// TIA Portal V17 program export: 1 tag tables, 0 data types, 2 data blocks, 2 code blocks (in call order from the OBs), 3 instance data blocks

VAR_GLOBAL   // PLC tag table "Default tag table"
   clockInput AT %I0.0 : Bool;   // Clock generator input
   Tag_1 AT %ID1000 : DWord;
   Axe_1_Signal_A AT %Q0.2 : Bool;
   Axe_1_Signal_B AT %Q0.3 : Bool;
END_VAR

DATA_BLOCK "DataExample1"   // DB1
{ S7_Optimized_Access := 'TRUE' }
VERSION : 0.1
// stored: AutoNumber true, DBAccessibleFromOPCUA true, IsOnlyStoredInLoadMemory false, IsRetainMemResEnabled false, IsWriteProtectedInAS false, MemoryReserve 100
   VAR
      hscData { S7_SetPoint := 'True'} : HSC_Period;   // Instruction CTRL_HSC_EXT: CTRL
      hscDone : Bool;   // Instruction CTRL_HSC_EXT: Done
      hscBusy : Bool;   // Instruction CTRL_HSC_EXT: Busy
      hscError : Bool;   // Instruction CTRL_HSC_EXT: Error
      hscStatus : Word;   // Instruction CTRL_HSC_EXT: Status
      numPulsePerRot : Int := 1000;   // Number of pulses per rotation
      overflow : Bool;   // Elapsed time overflow
      speed : Real := 0.0;   // Calculated speed [rpm]
      vitesse : Real;
   END_VAR
BEGIN
   hscData.EnHSC := TRUE;
   hscData.NewPeriod := 10;
END_DATA_BLOCK

DATA_BLOCK "DataExample2"   // DB5
{ S7_Optimized_Access := 'TRUE' }
VERSION : 0.1
// stored: AutoNumber false, DBAccessibleFromOPCUA true, IsOnlyStoredInLoadMemory false, IsRetainMemResEnabled false, IsWriteProtectedInAS false, MemoryReserve 100
   VAR
      hscData { S7_SetPoint := 'True'} : HSC_Period;   // Instruction CTRL_HSC_EXT: CTRL
      hscDone : Bool;   // Instruction CTRL_HSC_EXT: Done
      hscBusy : Bool;   // Instruction CTRL_HSC_EXT: Busy
      hscError : Bool;   // Instruction CTRL_HSC_EXT: Error
      hscStatus : Word;   // Instruction CTRL_HSC_EXT: Status
      numPulsePerRot : Int := 1000;   // Number of pulses per rotation
      overflow : Bool;   // Elapsed time overflow
      speed : Real := 0.0;   // Calculated speed [rpm]
      vitesse : Real;
      hsc1 : HSC_Count;
   END_VAR
BEGIN
   hscData.EnHSC := TRUE;
   hscData.NewPeriod := 10;
END_DATA_BLOCK

ORGANIZATION_BLOCK "Main"   // OB1, FBD, ProgramCycle
TITLE = "Main Program Sweep (Cycle)"
{ S7_Optimized_Access := 'TRUE' }
VERSION : 0.1
// stored: AutoNumber true, IsIECCheckEnabled false, SetENOAutomatically false
   VAR_INPUT
      Initial_Call : Bool;   // Initial call of this OB
      Remanence : Bool;   // =True, if remanent data are available
   END_VAR
BEGIN

REGION Network 1: Call CTRL_HSC_EXT for HSC1
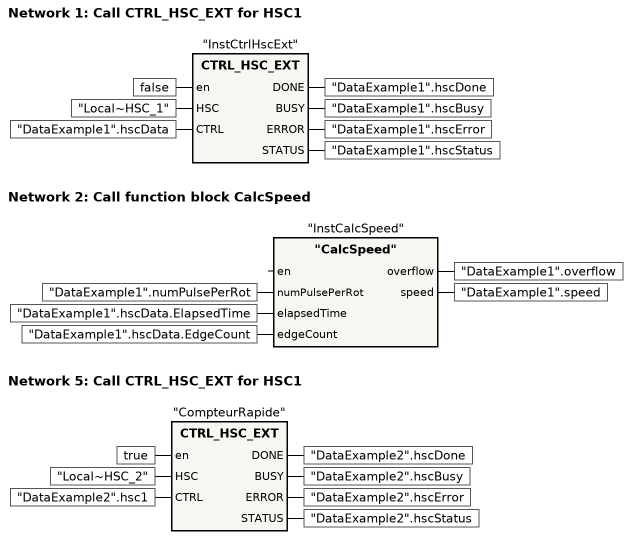
   IF false THEN
       "InstCtrlHscExt"(HSC := "Local~HSC_1",   // CTRL_HSC_EXT
                        CTRL := "DataExample1".hscData,
                        DONE => "DataExample1".hscDone,
                        BUSY => "DataExample1".hscBusy,
                        ERROR => "DataExample1".hscError,
                        STATUS => "DataExample1".hscStatus);
   END_IF;
END_REGION

REGION Network 2: Call function block CalcSpeed
   "InstCalcSpeed"(numPulsePerRot := "DataExample1".numPulsePerRot,   // "CalcSpeed"
                   elapsedTime := "DataExample1".hscData.ElapsedTime,
                   edgeCount := "DataExample1".hscData.EdgeCount,
                   overflow => "DataExample1".overflow,
                   speed => "DataExample1".speed);
END_REGION

REGION Network 3 (SCL)
   "DataExample1".vitesse := 0.2 * "DataExample1".speed;
END_REGION

REGION Network 5: Call CTRL_HSC_EXT for HSC1
   IF true THEN
       "CompteurRapide"(HSC := "Local~HSC_2",   // CTRL_HSC_EXT
                        CTRL := "DataExample2".hsc1,
                        DONE => "DataExample2".hscDone,
                        BUSY => "DataExample2".hscBusy,
                        ERROR => "DataExample2".hscError,
                        STATUS => "DataExample2".hscStatus);
   END_IF;
END_REGION
END_ORGANIZATION_BLOCK

FUNCTION_BLOCK "CalcSpeed"
{ S7_Optimized_Access := 'TRUE' }
VERSION : 0.1
   VAR_INPUT 
      numPulsePerRot : Int;
      elapsedTime { ExternalAccessible := 'False'; ExternalVisible := 'False'; ExternalWritable := 'False'} : UDInt;
      edgeCount { ExternalAccessible := 'False'; ExternalVisible := 'False'; ExternalWritable := 'False'} : UDInt;
   END_VAR

   VAR_OUTPUT 
      overflow { ExternalWritable := 'False'} : Bool;
      speed { ExternalWritable := 'False'} : Real;
   END_VAR

   VAR 
      statPeriod { ExternalAccessible := 'False'; ExternalVisible := 'False'; ExternalWritable := 'False'} : Real;
      statOverflow { ExternalAccessible := 'False'; ExternalVisible := 'False'; ExternalWritable := 'False'} : Bool;
   END_VAR

   VAR CONSTANT 
      BILLION : Real := 1.0E+09;
      OVERFLOW_VALUE : UDInt := 4294967295;
   END_VAR


BEGIN
	//=============================================================================
	//SIEMENS AG
	//(c)Copyright 2016 All Rights Reserved
	//-----------------------------------------------------------------------------
	//Library:       -
	//Tested with:   S7-1200 V4.2
	//Engineering:   TIA Portal V14
	//Restrictions:  -
	//Requirements:  S7-1200
	//Functionality: Basic axis functions, as power, reset, home and jog
	//-----------------------------------------------------------------------------
	//Change log table:
	//Version  Date       Expert in charge Changes applied
	//01.00.00 09.11.2016 Online Support   First released version
	//=============================================================================
	
	// #elapsedTime (range): 0 to 4.294.967.280
	// #elapsedTime (overflow): 4.294.967.295 (0xFFFF FFFF)
	
	// If EdgeCount and ElapsedTime is valid, calculate the period
	IF (#edgeCount > 0)
	  AND (#elapsedTime > 0)
	  AND (#elapsedTime <= 4294967280)
	THEN
	  // Calculate the period in nanoseconds 
	  #statPeriod := #elapsedTime / #edgeCount;
	  // Calculate the period in seconds 
	  #statPeriod := #numPulsePerRot * #statPeriod / #BILLION;
	END_IF;
	
	// Check overflow (the period between two pulse edges exceeds 4.295 seconds)
	IF (#elapsedTime = #OVERFLOW_VALUE)
	THEN
	  #statOverflow := TRUE;
	ELSE
	  #statOverflow := FALSE;
	END_IF;
	
	// Set period to zero, if overflow
	IF(#statOverflow = TRUE)
	THEN
	  #statPeriod := 0;
	END_IF;
	
	// Calculate speed in rpm
	IF (#statPeriod > 0)
	THEN
	  #speed := 1 / #statPeriod * 60.0;
	ELSE
	  #speed := 0;
	END_IF;
	
	// Set output overflow
	#overflow := #statOverflow;
	
END_FUNCTION_BLOCK

DATA_BLOCK "InstCalcSpeed"   // DB3
VERSION : 0.1
// stored: AutoNumber true, DBAccessibleFromOPCUA true, InstanceOfName CalcSpeed, InstanceOfType FB
"CalcSpeed"
BEGIN
END_DATA_BLOCK

DATA_BLOCK "CompteurRapide"   // DB4
// stored: AutoNumber true, DBAccessibleFromOPCUA true, InstanceOfName HSC, OfSystemLibElement CTRL_HSC_EXT, OfSystemLibVersion 1.0
"HSC"
   // VAR_INPUT
   //    HSC : HW_HSC;
   // END_VAR
   // VAR_OUTPUT
   //    DONE : Bool;
   //    BUSY : Bool;
   //    ERROR : Bool;
   //    STATUS : Word;
   // END_VAR
   // VAR_IN_OUT
   //    CTRL : Variant;
   // END_VAR
BEGIN
END_DATA_BLOCK

DATA_BLOCK "InstCtrlHscExt"   // DB2
// stored: AutoNumber true, DBAccessibleFromOPCUA true, InstanceOfName HSC, OfSystemLibElement CTRL_HSC_EXT, OfSystemLibVersion 1.0
"HSC"
   // VAR_INPUT
   //    HSC : HW_HSC;
   // END_VAR
   // VAR_OUTPUT
   //    DONE : Bool;
   //    BUSY : Bool;
   //    ERROR : Bool;
   //    STATUS : Word;
   // END_VAR
   // VAR_IN_OUT
   //    CTRL : Variant;
   // END_VAR
BEGIN
END_DATA_BLOCK
